FUNCTION_BLOCK E_SREN (* Event-driven quad-state *)
  (* Standard: 61499-1 Annex A; Description: Copyright (c), HR Agrartechnik GmbH This program and the accompanying materials are made available under the terms of the Eclipse Public License 2.0 which is available at https://www.eclipse.org/legal/epl-2.0/ SPDX-License-Identifier: EPL-2.0 The Output Q will be TRUE only at S. The Output Q will be FALSE only at R and ERR. The Output Q will be not changed at NONE *)
  PACKAGE logiBUS::utils::quarter;
  IMPORT logiBUS::utils::quarter::const::quarter;
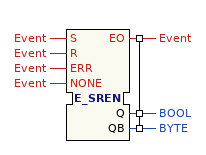
  EVENT_INPUT
    S; (* Enabled (on, active, etc.) *)
    R; (* Disabled (off, passive, etc.) *)
    ERR; (* Error indicator *)
    NONE; (* Not available or not installed *)
  END_EVENT
  EVENT_OUTPUT
    EO WITH Q, QB; (* Output Q has changed *)
  END_EVENT
  VAR_OUTPUT
    Q : BOOL := FALSE; (* BOOL Output *)
    QB : BYTE := quarter::COMMAND_DISABLE; (* 2bit (quarter Byte) Output with 4 States *)
  END_VAR
  VAR
    old_Q : BOOL := FALSE; (* old BOOL Output *)
    old_QB : BYTE := quarter::COMMAND_DISABLE; (* old 2bit (quarter Byte) Output with 4 States *)
  END_VAR
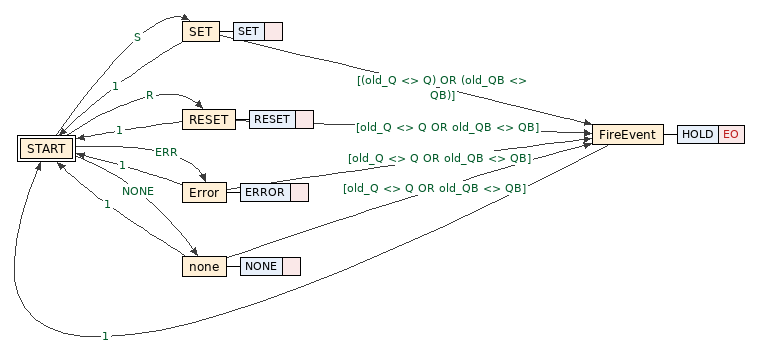
  EC_STATES
    START; (* Initial State *)
    SET : SET;
    RESET : RESET;
    Error : ERROR;
    none : NONE;
    FireEvent : HOLD -> EO;
  END_STATES
  EC_TRANSITIONS
    START TO SET := S;
    START TO RESET := R;
    START TO Error := ERR;
    SET TO FireEvent := [(old_Q <> Q) OR (old_QB <> QB)];
    RESET TO FireEvent := [old_Q <> Q OR old_QB <> QB];
    Error TO FireEvent := [old_Q <> Q OR old_QB <> QB];
    none TO FireEvent := [old_Q <> Q OR old_QB <> QB];
    FireEvent TO START := 1;
    SET TO START := 1;
    RESET TO START := 1;
    Error TO START := 1;
    none TO START := 1;
    START TO none := NONE;
  END_TRANSITIONS
  ALGORITHM SET IN ST:
Q := TRUE;
QB := quarter::COMMAND_ENABLE;
  END_ALGORITHM
  ALGORITHM RESET IN ST:
Q := FALSE;
QB := quarter::COMMAND_DISABLE;
  END_ALGORITHM
  ALGORITHM ERROR IN ST:
Q := FALSE;
QB := quarter::STATUS_ERROR;
  END_ALGORITHM
  ALGORITHM NONE IN ST:
// Q Don't care/take no action (leave function as is)
QB := quarter::COMMAND_NO_ACTION;
  END_ALGORITHM
  ALGORITHM HOLD IN ST:
old_Q := Q;
old_QB := QB;
  END_ALGORITHM
END_FUNCTION_BLOCK
